TYPE udt_ECAT_NodeImage_20200618 :
STRUCT
	sType:STRING;
	
END_STRUCT
END_TYPE

(* stored: Version 1.1.0.1, ProductVersion 3.1.4024.4
   DUT udt_ECAT_NodeImage_20200618: Id {f73079c7-f42f-4461-b75f-f234dba01d43} *)
